(* Logix 5000 project; controller new_PLC_1 vendor 1 type 14 code 235 rev 37.11; software revision 37.00 *)

TASK MainTask (continuous, watchdog 500 ms) : MainProgram
TASK SafetyTask (periodic, rate 20 ms, priority 10, watchdog 20 ms, safety) : SafetyProgram

MODULES
   Local : vendor 1 type 14 code 235 (5069 0, rev 37.11)
      Tarjeta_Ethernet : vendor 1 type 12 code 200 (Ethernet 10.12.143.10, rev 10.7, Output RPI 10 ms)
         PLC_Safety : vendor 1 type 14 code 148 (ICP 1, rev 31.11, $66e82ebd$ RPI 20 ms)
         @7686e93b@:Partner : vendor 1 type 14 code 146 (ICP 2, rev 31.11)
      Variador_Conveyor_1 : PowerFlex 525-EENET (Ethernet 10.12.143.6, rev 5.1, Output RPI 20 ms)
      Camera_Conveyor_1 : vendor 678 type 100 code 260 (Ethernet 10.12.143.5, rev 12.1, Output RPI 60 ms)
      Point_IO_Gabinete_1 : 1734-AENTR (Ethernet 10.12.143.40, rev 5.12, Output RPI 20 ms)
         Modulo_Input_11 : 1734-IB8 (PointIO 1, rev 3.22)
              Point_IO_Gabinete_1:1:I.0   // Sensor Axis X -
              Point_IO_Gabinete_1:1:I.1   // Sensor Axis X +
              Point_IO_Gabinete_1:1:I.2   // Sensor Gripper Turn Conveyor
              Point_IO_Gabinete_1:1:I.3   // Sensor Gripper Close
              Point_IO_Gabinete_1:1:I.4   // Sensor Gripper Turn Storage
              Point_IO_Gabinete_1:1:I.5   // Sensor Axis Y -
              Point_IO_Gabinete_1:1:I.6   // Sensor Axis Y +
              Point_IO_Gabinete_1:1:I.7   // Sensor Gripper Open
              Point_IO_Gabinete_1:1:I   // Storage 1 Inputs
         Modulo_Input_12 : 1734-IB8 (PointIO 2, rev 3.22)
         Modulo_Output_11 : 1734-OB8 (PointIO 3, rev 3.22)
              Point_IO_Gabinete_1:3:O.0   // Axis X +
              Point_IO_Gabinete_1:3:O.1   // Axis X -
              Point_IO_Gabinete_1:3:O.2   // Gripper Close
              Point_IO_Gabinete_1:3:O.3   // Gripper Open
              Point_IO_Gabinete_1:3:O.4   // Gripper Turn Conveyor
              Point_IO_Gabinete_1:3:O.5   // Gripper Turn Storage
              Point_IO_Gabinete_1:3:O.6   // Axis Y +
              Point_IO_Gabinete_1:3:O.7   // Axis Y -
              Point_IO_Gabinete_1:3:O   // Storage 1 Outputs
         Modulo_Output_12 : 1734-OB8 (PointIO 4, rev 3.22)
              Point_IO_Gabinete_1:4:O.0   // Stack Light Blue
              Point_IO_Gabinete_1:4:O.1   // Stack Light Green
              Point_IO_Gabinete_1:4:O.2   // Stack Light Orange
              Point_IO_Gabinete_1:4:O.3   // Stack Light Red
              Point_IO_Gabinete_1:4:O   // Storage 1 Outputs Stack Lights
         Modulo_Relay_1 : 1734-OW4 (PointIO 5, rev 3.22)
      Point_IO_Gabinete_3 : 1734-AENTR (Ethernet 10.12.143.42, rev 5.12, Output RPI 20 ms)
         Modulo_Input_31 : 1734-IB8 (PointIO 1, rev 3.22)
         Modulo_Input_32 : 1734-IB8 (PointIO 2, rev 3.22)
         Modulo_Input_33 : 1734-IB8 (PointIO 3, rev 3.22)
              Point_IO_Gabinete_3:3:I.4   // Sensor Lane Change 2 +
              Point_IO_Gabinete_3:3:I.6   // Sensor Lane Change 1 +
              Point_IO_Gabinete_3:3:I.2   // Piston 1 retraido conveyor 1
              Point_IO_Gabinete_3:3:I.3   // Piston 1 activado conveyor 1
              Point_IO_Gabinete_3:3:I   // Sensors Lane Change +
         Modulo_Input_34 : 1734-IB8 (PointIO 4, rev 3.22)
              Point_IO_Gabinete_3:4:I.0   // Sensor Lane Change 1 -
              Point_IO_Gabinete_3:4:I.4   // Sensor Lane Change 2 -
              Point_IO_Gabinete_3:4:I   // Sensors Lane Change -
         Modulo_Input_35 : 1734-IB8 (PointIO 5, rev 3.22)
              Point_IO_Gabinete_3:5:I.0   // Inductive Sensor 1
              Point_IO_Gabinete_3:5:I.1   // Inductive Sensor 6
              Point_IO_Gabinete_3:5:I.2   // Inductive Sensor 5
              Point_IO_Gabinete_3:5:I.3   // Inductive Sensor 4
              Point_IO_Gabinete_3:5:I.4   // Inductive Sensor 3
              Point_IO_Gabinete_3:5:I.5   // Inductive Sensor 2
              Point_IO_Gabinete_3:5:I   // Conveyor 1 Inductive Sensors
         Modulo_Input_36 : 1734-IB8 (PointIO 6, rev 3.22)
         Modulo_Output_31 : 1734-OB8 (PointIO 7, rev 3.22)
              Point_IO_Gabinete_3:7:O.0   // Pneumatic Cylinder 0
              Point_IO_Gabinete_3:7:O.1   // Pneumatic Cylinder 1
              Point_IO_Gabinete_3:7:O.2   // Pneumatic Cylinder 2
              Point_IO_Gabinete_3:7:O.3   // Pneumatic Cylinder 3
              Point_IO_Gabinete_3:7:O.4   // Pneumatic Cylinder 4
              Point_IO_Gabinete_3:7:O.5   // Pneumatic Cylinder D
              Point_IO_Gabinete_3:7:O.6   // Lane Change 2
              Point_IO_Gabinete_3:7:O.7   // Lane Change 1
              Point_IO_Gabinete_3:7:O   // Conveyor 1 Pneumatic Cylinders
         Modulo_Output_32 : 1734-OB8 (PointIO 8, rev 3.22)
              Point_IO_Gabinete_3:8:O.0   // Main Valve
              Point_IO_Gabinete_3:8:O.2   // Cognex Light 2
              Point_IO_Gabinete_3:8:O.3   // Cognex Light 1
              Point_IO_Gabinete_3:8:O   // Main Valve
         Modulo_Relay_31 : 1734-OW4 (PointIO 9, rev 3.22)
         Modulo_Relay_32 : 1734-OW4 (PointIO 10, rev 3.22)
      PLC2 : vendor 1 type 14 code 235 (Ethernet 10.12.143.18, rev 37.11, $66dc2b48$ RPI 20 ms)
END_MODULES

VAR_GLOBAL   (* controller tags *)
   Data_from_PLC_2 : DINT[20];
   Data_From_PLC_Safety : DINT[20] := ([1] := 128);
        [0].11   // Pieza 1 puesta
        [0].12   // Pieza 2 puesta
        [0].13   // Pieza 3 puesta
        [0].14   // Pieza1 dejada
        [0].15   // Pieza 2 dejada
        [0].17   // Pieza 3 dejada
   Data_to_PLC_2 : DINT[20]; {produced}
        [0].0   // PB_START CONVEYORS DE PLC1 Y PLC2
        [1].0   // Pieza 1 etapa 1 salida y recorrido
        [1].1   // Pieza 1 etapa 2 foto cognex
        [1].2   // Pieza 1 etapa 3 listo para recolección
        [1].5   // Pieza 2 etapa 2 foto cognex
        [1].6   // Pieza 2 etapa 3 listo para recolección
        [1].8   // Pieza 3 etapa 2 foto cognex
        [1].7   // Pieza 3 etapa 1 salida y recorrido
        [1].4   // Pieza 2 etapa 1 salida y recorrido
        [1].9   // Pieza 3 etapa 3 listo para recolección
   Data_To_PLC_Safety : DINT[20] := ([0] := 16777216); {produced}
        [19].0   // Dato para mandar el trigger
   Fanuc_Strobe : BOOL;
   Height_1 : BOOL;
   Height_2 : BOOL;
   Height_3 : BOOL;
   Height_4 : BOOL;
   Height_5 : BOOL;
   Height_6 : BOOL;
   Height_Conveyor_1 : BOOL;
   Height_Conveyor_2 : BOOL;
   Process_1_Reset : ALIAS FOR Point_IO_Gabinete_1:2:I.6;   // Push Button Process 1 Reset
   Safety_OK : BOOL;
   Sensor_Height_1 : BOOL;
   Sensor_Height_2 : BOOL;
   Sensor_Height_3 : BOOL;
   Sensor_Height_4 : BOOL;
   Sensor_Height_5 : BOOL;
   Sensor_Height_6 : BOOL;
   Sensor_Height_Conveyor_1 : BOOL;
   Sensor_Height_Conveyor_2 : BOOL;
   Storage_On : BOOL;
END_VAR

PROGRAM MainProgram   (* main routine MainRoutine *)
VAR
   cleaning : BOOL;
   Counter_1 : COUNTER := (PRE := 3);
   Height_4_Number_2 : BOOL;
   Height_5_Number_2 : BOOL;
   Height_6_Number_2 : BOOL;
   HMI_Conveyor_OFF : BOOL;
   HMI_Conveyor_ON : BOOL;
   HMI_Fcognex1 : BOOL := 1;
   HMI_Fpowerflex1 : BOOL;
   HMI_Gripper_Close : BOOL;
   HMI_Gripper_Open : BOOL;
   HMI_Height_4_1 : BOOL;
   HMI_Height_4_2 : BOOL;
   HMI_Height_5_1 : BOOL;
   HMI_Height_5_2 : BOOL;
   HMI_Height_6_1 : BOOL;
   HMI_Height_6_2 : BOOL;
   HMI_Lane_Change_1 : BOOL;
   HMI_Lane_Change_2 : BOOL;
   HMI_Pneumatic_Cylinder_0 : BOOL;
   HMI_Pneumatic_Cylinder_1 : BOOL;
   HMI_Pneumatic_Cylinder_2 : BOOL;
   HMI_Pneumatic_Cylinder_3 : BOOL;
   HMI_Pneumatic_Cylinder_4 : BOOL;
   HMi_Screen_Storage1 : BOOL := 1;
   HMI_Turn_Conveyor : BOOL;
   HMI_Turn_Storage : BOOL;
   HMI_Y_Negative : BOOL;
   HMI_Y_Positive : BOOL;
   Pieza : COUNTER := (PRE := 3);
   Pieza_Detectada : BOOL;
   Pneumatic_Cylinder_0 : ALIAS FOR Point_IO_Gabinete_3:7:O.0;
   Recieve_bit_From_FANUC : BOOL;
   Reset_manual : BOOL;
   Send_Bit_to_FANUC_1 : BOOL;
   Send_Bit_to_FANUC_2 : BOOL;
   Send_Bit_to_FANUC_3 : BOOL;
   Send_Bit_to_FANUC_4 : BOOL;
   Sensor_Height_4_Number_2 : BOOL;
   Sensor_Height_5_Number_2 : BOOL;
   Sensor_Height_6_Number_2 : BOOL;
   Start_Button_1 : BOOL;
   Start_Button_2 : BOOL;
   Start_Button_3 : BOOL;
   Start_Conveyor1 : BOOL;
   Start_Robot_Fanuc : BOOL;
   Step_000 : SFC_STEP := (Status := 16#0020_0000, PauseTimer := 1);
   Step_001 : SFC_STEP := (Status := 16#0020_0000, PauseTimer := 1);
   Tiempo_ciclo : TIMER := (PRE := 1000000);
   Timer1 : TIMER := (PRE := 1000);
   Timer2 : TIMER := (PRE := 1000);
   Timer3 : TIMER := (PRE := 15000);
   Timer4 : TIMER := (PRE := 2000);
   Timer5 : TIMER := (PRE := 2000);
   Timer6 : TIMER := (PRE := 1000);
   Timer7 : TIMER := (PRE := 2000);
   Timer8 : TIMER := (PRE := 2000);
   timer_counter_1 : TIMER := (PRE := 2000);
   Timer_trigger : TIMER := (PRE := 3000);
   Tran_000 : BOOL;
   Tran_001 : BOOL;
   Trigger_Cognex_3 : BOOL;
END_VAR

ROUTINE E_Stop   (* ladder *)
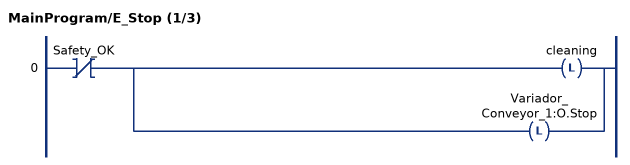
   0: XIO(Safety_OK)[OTL(cleaning) ,OTL(Variador_Conveyor_1:O.Stop) ];
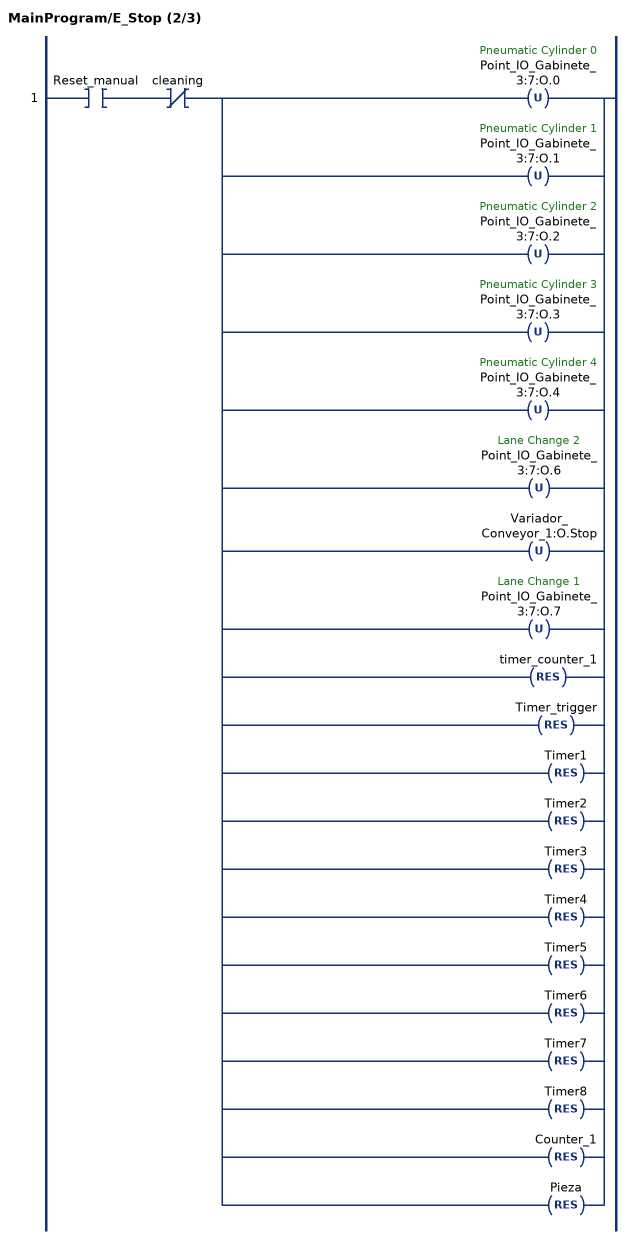
   1: XIC(Reset_manual)XIO(cleaning)[OTU(Point_IO_Gabinete_3:7:O.0) ,OTU(Point_IO_Gabinete_3:7:O.1) ,OTU(Point_IO_Gabinete_3:7:O.2) ,OTU(Point_IO_Gabinete_3:7:O.3) ,OTU(Point_IO_Gabinete_3:7:O.4) ,OTU(Point_IO_Gabinete_3:7:O.6) ,OTU(Variador_Conveyor_1:O.Stop) ,OTU(Point_IO_Gabinete_3:7:O.7) ,RES(timer_counter_1) ,RES(Timer_trigger) ,RES(Timer1) ,RES(Timer2) ,RES(Timer3) ,RES(Timer4) ,RES(Timer5) ,RES(Timer6) ,RES(Timer7) ,RES(Timer8) ,RES(Counter_1) ,RES(Pieza) ];
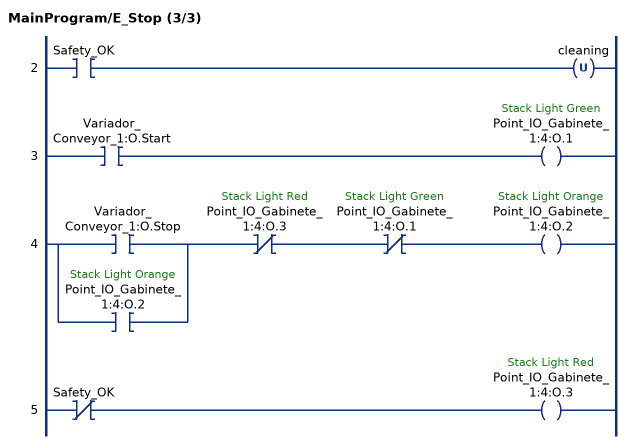
   2: XIC(Safety_OK)OTU(cleaning);
   3: XIC(Variador_Conveyor_1:O.Start)OTE(Point_IO_Gabinete_1:4:O.1);
   4: [XIC(Variador_Conveyor_1:O.Stop) ,XIC(Point_IO_Gabinete_1:4:O.2) ]XIO(Point_IO_Gabinete_1:4:O.3)XIO(Point_IO_Gabinete_1:4:O.1)OTE(Point_IO_Gabinete_1:4:O.2);
   5: XIO(Safety_OK)OTE(Point_IO_Gabinete_1:4:O.3);
END_ROUTINE

ROUTINE MainRoutine   (* ladder *)
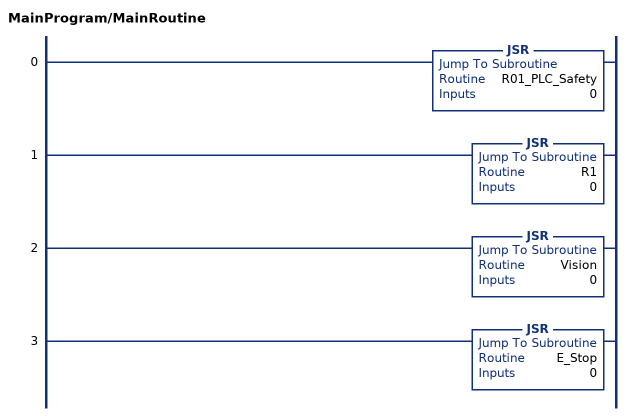
   0: JSR(R01_PLC_Safety,0);
   1: JSR(R1,0);
   2: JSR(Vision,0);
   3: JSR(E_Stop,0);
END_ROUTINE

ROUTINE R01_PLC_Safety   (* ladder *)
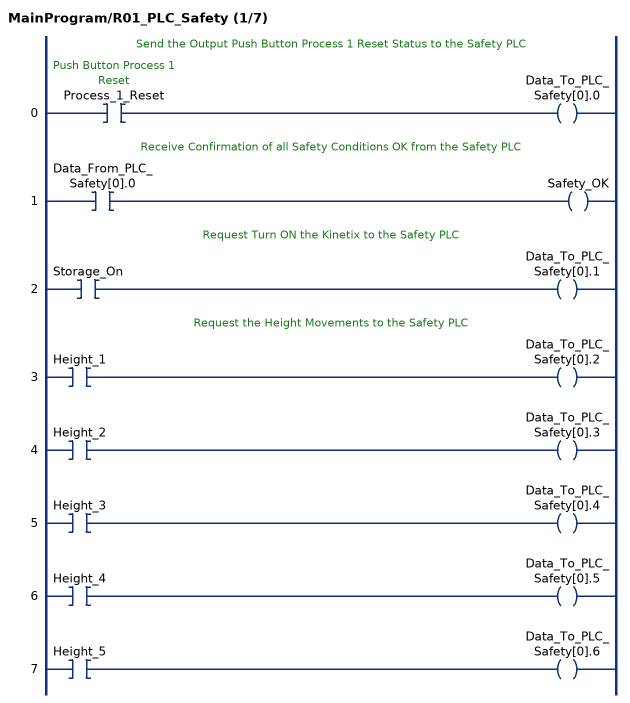
   // Send the Output Push Button Process 1 Reset Status to the Safety PLC
   0: XIC(Process_1_Reset)OTE(Data_To_PLC_Safety[0].0);
   // Receive Confirmation of all Safety Conditions OK from the Safety PLC
   1: XIC(Data_From_PLC_Safety[0].0)OTE(Safety_OK);
   // Request Turn ON the Kinetix to the Safety PLC
   2: XIC(Storage_On)OTE(Data_To_PLC_Safety[0].1);
   // Request the Height Movements to the Safety PLC
   3: XIC(Height_1)OTE(Data_To_PLC_Safety[0].2);
   4: XIC(Height_2)OTE(Data_To_PLC_Safety[0].3);
   5: XIC(Height_3)OTE(Data_To_PLC_Safety[0].4);
   6: XIC(Height_4)OTE(Data_To_PLC_Safety[0].5);
   7: XIC(Height_5)OTE(Data_To_PLC_Safety[0].6);
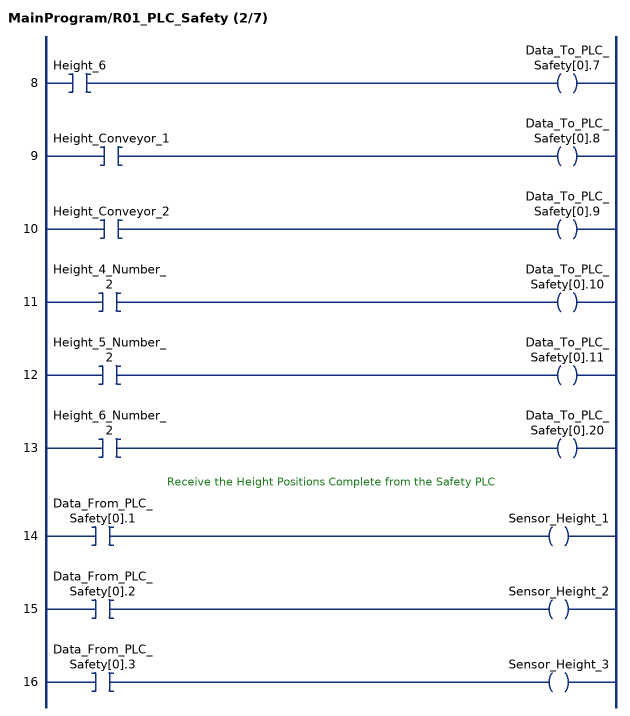
   8: XIC(Height_6)OTE(Data_To_PLC_Safety[0].7);
   9: XIC(Height_Conveyor_1)OTE(Data_To_PLC_Safety[0].8);
   10: XIC(Height_Conveyor_2)OTE(Data_To_PLC_Safety[0].9);
   11: XIC(Height_4_Number_2)OTE(Data_To_PLC_Safety[0].10);
   12: XIC(Height_5_Number_2)OTE(Data_To_PLC_Safety[0].11);
   13: XIC(Height_6_Number_2)OTE(Data_To_PLC_Safety[0].20);
   // Receive the Height Positions Complete from the Safety PLC
   14: XIC(Data_From_PLC_Safety[0].1)OTE(Sensor_Height_1);
   15: XIC(Data_From_PLC_Safety[0].2)OTE(Sensor_Height_2);
   16: XIC(Data_From_PLC_Safety[0].3)OTE(Sensor_Height_3);
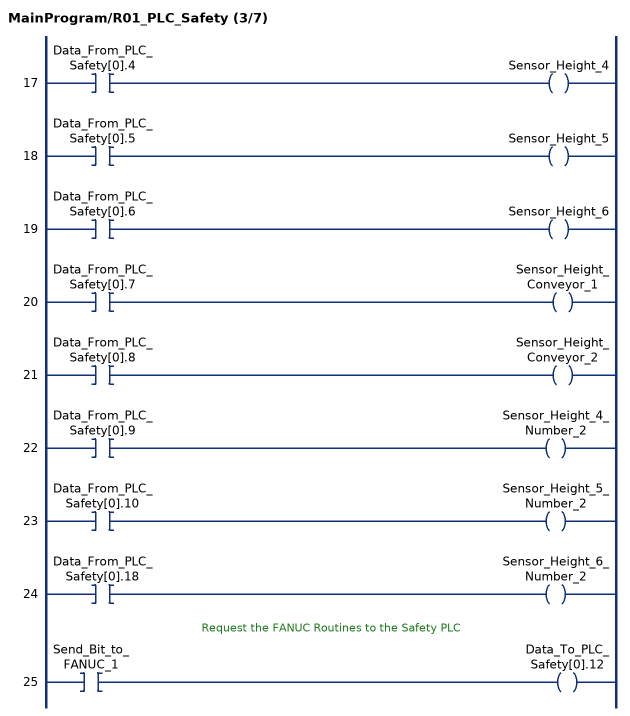
   17: XIC(Data_From_PLC_Safety[0].4)OTE(Sensor_Height_4);
   18: XIC(Data_From_PLC_Safety[0].5)OTE(Sensor_Height_5);
   19: XIC(Data_From_PLC_Safety[0].6)OTE(Sensor_Height_6);
   20: XIC(Data_From_PLC_Safety[0].7)OTE(Sensor_Height_Conveyor_1);
   21: XIC(Data_From_PLC_Safety[0].8)OTE(Sensor_Height_Conveyor_2);
   22: XIC(Data_From_PLC_Safety[0].9)OTE(Sensor_Height_4_Number_2);
   23: XIC(Data_From_PLC_Safety[0].10)OTE(Sensor_Height_5_Number_2);
   24: XIC(Data_From_PLC_Safety[0].18)OTE(Sensor_Height_6_Number_2);
   // Request the FANUC Routines to the Safety PLC
   25: XIC(Send_Bit_to_FANUC_1)OTE(Data_To_PLC_Safety[0].12);
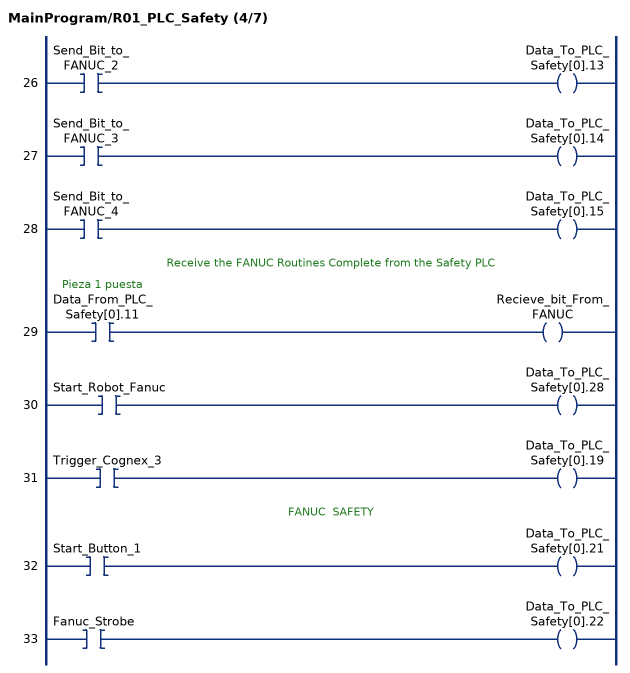
   26: XIC(Send_Bit_to_FANUC_2)OTE(Data_To_PLC_Safety[0].13);
   27: XIC(Send_Bit_to_FANUC_3)OTE(Data_To_PLC_Safety[0].14);
   28: XIC(Send_Bit_to_FANUC_4)OTE(Data_To_PLC_Safety[0].15);
   // Receive the FANUC Routines Complete from the Safety PLC
   29: XIC(Data_From_PLC_Safety[0].11)OTE(Recieve_bit_From_FANUC);
   30: XIC(Start_Robot_Fanuc)OTE(Data_To_PLC_Safety[0].28);
   31: XIC(Trigger_Cognex_3)OTE(Data_To_PLC_Safety[0].19);
   // FANUC  SAFETY
   32: XIC(Start_Button_1)OTE(Data_To_PLC_Safety[0].21);
   33: XIC(Fanuc_Strobe)OTE(Data_To_PLC_Safety[0].22);
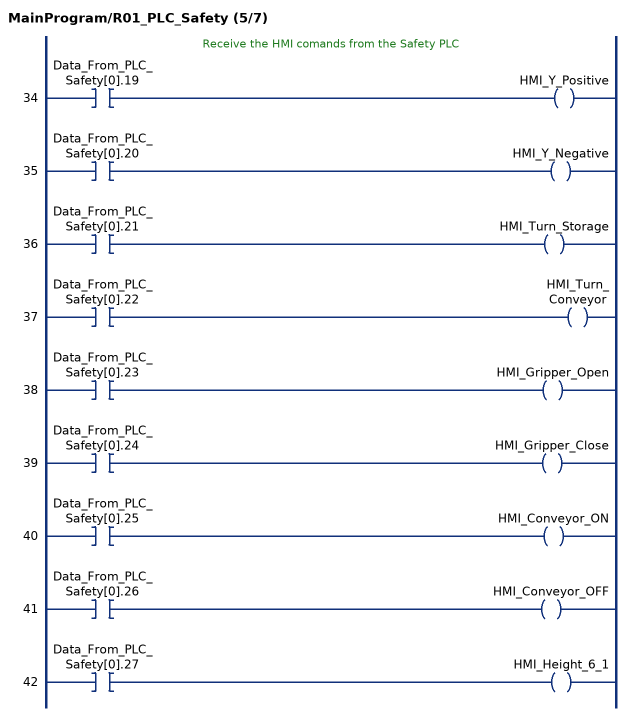
   // Receive the HMI comands from the Safety PLC
   34: XIC(Data_From_PLC_Safety[0].19)OTE(HMI_Y_Positive);
   35: XIC(Data_From_PLC_Safety[0].20)OTE(HMI_Y_Negative);
   36: XIC(Data_From_PLC_Safety[0].21)OTE(HMI_Turn_Storage);
   37: XIC(Data_From_PLC_Safety[0].22)OTE(HMI_Turn_Conveyor);
   38: XIC(Data_From_PLC_Safety[0].23)OTE(HMI_Gripper_Open);
   39: XIC(Data_From_PLC_Safety[0].24)OTE(HMI_Gripper_Close);
   40: XIC(Data_From_PLC_Safety[0].25)OTE(HMI_Conveyor_ON);
   41: XIC(Data_From_PLC_Safety[0].26)OTE(HMI_Conveyor_OFF);
   42: XIC(Data_From_PLC_Safety[0].27)OTE(HMI_Height_6_1);
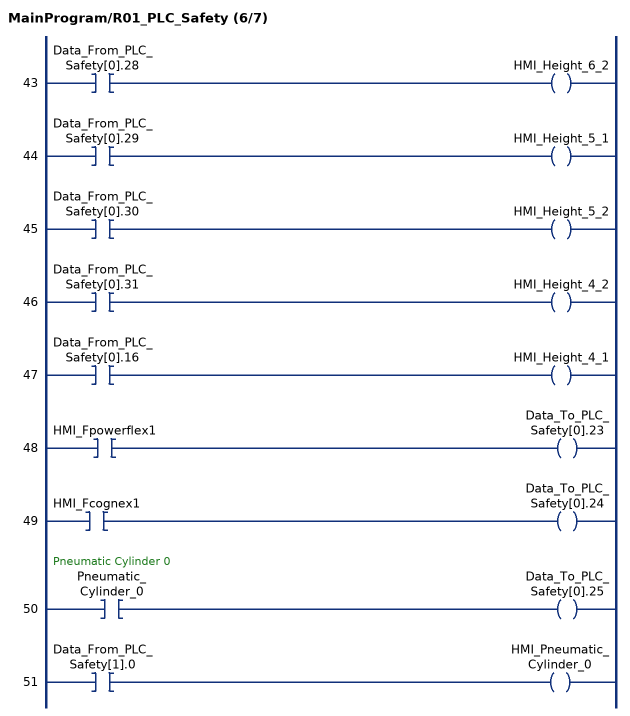
   43: XIC(Data_From_PLC_Safety[0].28)OTE(HMI_Height_6_2);
   44: XIC(Data_From_PLC_Safety[0].29)OTE(HMI_Height_5_1);
   45: XIC(Data_From_PLC_Safety[0].30)OTE(HMI_Height_5_2);
   46: XIC(Data_From_PLC_Safety[0].31)OTE(HMI_Height_4_2);
   47: XIC(Data_From_PLC_Safety[0].16)OTE(HMI_Height_4_1);
   48: XIC(HMI_Fpowerflex1)OTE(Data_To_PLC_Safety[0].23);
   49: XIC(HMI_Fcognex1)OTE(Data_To_PLC_Safety[0].24);
   50: XIC(Pneumatic_Cylinder_0)OTE(Data_To_PLC_Safety[0].25);
   51: XIC(Data_From_PLC_Safety[1].0)OTE(HMI_Pneumatic_Cylinder_0);
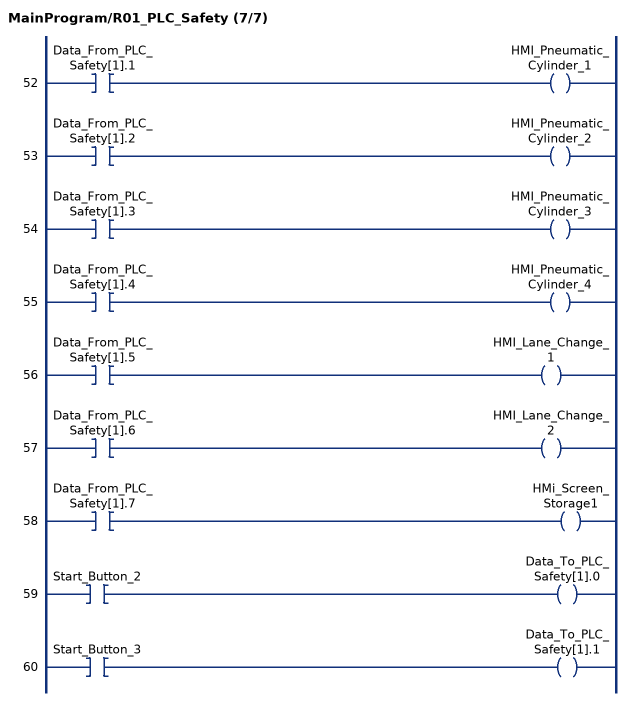
   52: XIC(Data_From_PLC_Safety[1].1)OTE(HMI_Pneumatic_Cylinder_1);
   53: XIC(Data_From_PLC_Safety[1].2)OTE(HMI_Pneumatic_Cylinder_2);
   54: XIC(Data_From_PLC_Safety[1].3)OTE(HMI_Pneumatic_Cylinder_3);
   55: XIC(Data_From_PLC_Safety[1].4)OTE(HMI_Pneumatic_Cylinder_4);
   56: XIC(Data_From_PLC_Safety[1].5)OTE(HMI_Lane_Change_1);
   57: XIC(Data_From_PLC_Safety[1].6)OTE(HMI_Lane_Change_2);
   58: XIC(Data_From_PLC_Safety[1].7)OTE(HMi_Screen_Storage1);
   59: XIC(Start_Button_2)OTE(Data_To_PLC_Safety[1].0);
   60: XIC(Start_Button_3)OTE(Data_To_PLC_Safety[1].1);
END_ROUTINE

ROUTINE R1   (* ladder *)
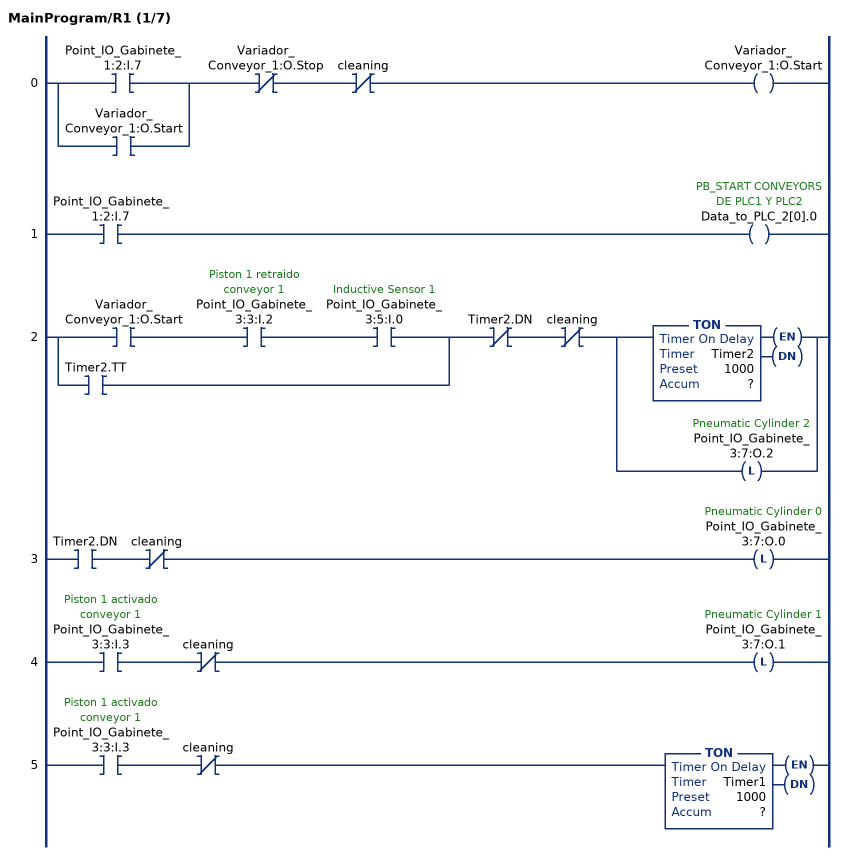
   0: [XIC(Point_IO_Gabinete_1:2:I.7) ,XIC(Variador_Conveyor_1:O.Start) ]XIO(Variador_Conveyor_1:O.Stop)XIO(cleaning)OTE(Variador_Conveyor_1:O.Start);
   1: XIC(Point_IO_Gabinete_1:2:I.7)OTE(Data_to_PLC_2[0].0);
   2: [XIC(Variador_Conveyor_1:O.Start) XIC(Point_IO_Gabinete_3:3:I.2) XIC(Point_IO_Gabinete_3:5:I.0) ,XIC(Timer2.TT) ]XIO(Timer2.DN)XIO(cleaning)[TON(Timer2,?,?) ,OTL(Point_IO_Gabinete_3:7:O.2) ];
   3: XIC(Timer2.DN)XIO(cleaning)OTL(Point_IO_Gabinete_3:7:O.0);
   4: XIC(Point_IO_Gabinete_3:3:I.3)XIO(cleaning)OTL(Point_IO_Gabinete_3:7:O.1);
   5: XIC(Point_IO_Gabinete_3:3:I.3)XIO(cleaning)TON(Timer1,?,?);
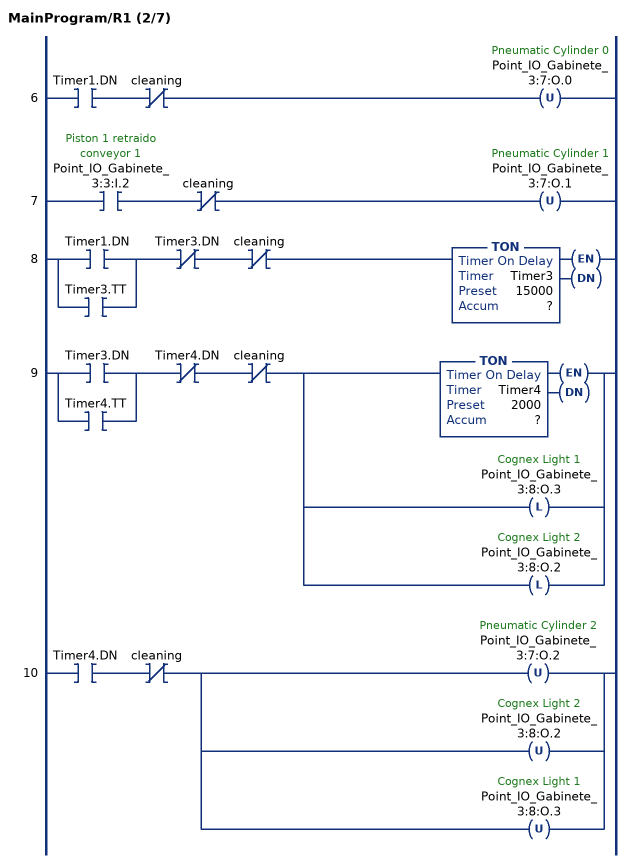
   6: XIC(Timer1.DN)XIO(cleaning)OTU(Point_IO_Gabinete_3:7:O.0);
   7: XIC(Point_IO_Gabinete_3:3:I.2)XIO(cleaning)OTU(Point_IO_Gabinete_3:7:O.1);
   8: [XIC(Timer1.DN) ,XIC(Timer3.TT) ]XIO(Timer3.DN)XIO(cleaning)TON(Timer3,?,?);
   9: [XIC(Timer3.DN) ,XIC(Timer4.TT) ]XIO(Timer4.DN)XIO(cleaning)[TON(Timer4,?,?) ,OTL(Point_IO_Gabinete_3:8:O.3) ,OTL(Point_IO_Gabinete_3:8:O.2) ];
   10: XIC(Timer4.DN)XIO(cleaning)[OTU(Point_IO_Gabinete_3:7:O.2) ,OTU(Point_IO_Gabinete_3:8:O.2) ,OTU(Point_IO_Gabinete_3:8:O.3) ];
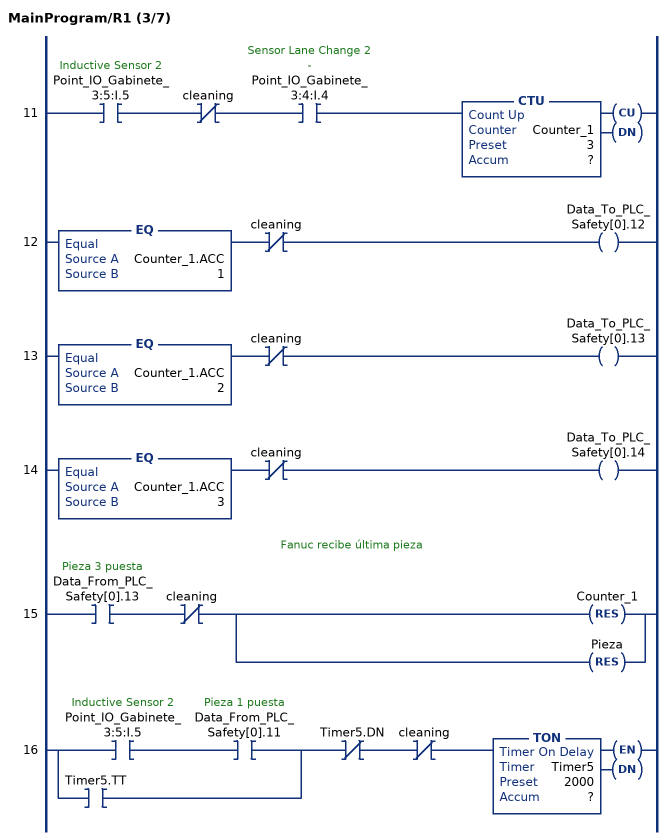
   11: XIC(Point_IO_Gabinete_3:5:I.5)XIO(cleaning)XIC(Point_IO_Gabinete_3:4:I.4)CTU(Counter_1,?,?);
   12: EQ(Counter_1.ACC,1)XIO(cleaning)OTE(Data_To_PLC_Safety[0].12);
   13: EQ(Counter_1.ACC,2)XIO(cleaning)OTE(Data_To_PLC_Safety[0].13);
   14: EQ(Counter_1.ACC,3)XIO(cleaning)OTE(Data_To_PLC_Safety[0].14);
   // Fanuc recibe última pieza
   15: XIC(Data_From_PLC_Safety[0].13)XIO(cleaning)[RES(Counter_1) ,RES(Pieza) ];
   16: [XIC(Point_IO_Gabinete_3:5:I.5) XIC(Data_From_PLC_Safety[0].11) ,XIC(Timer5.TT) ]XIO(Timer5.DN)XIO(cleaning)TON(Timer5,?,?);
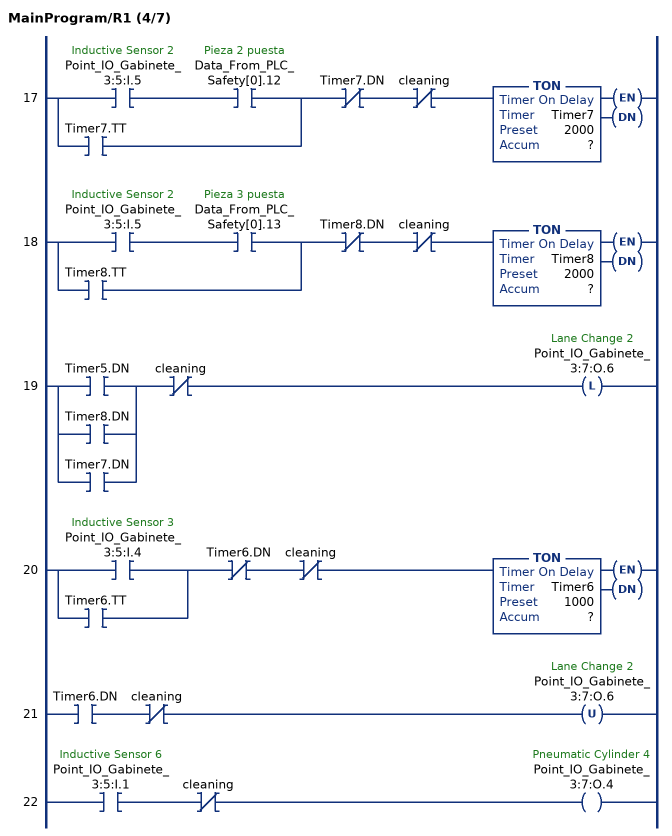
   17: [XIC(Point_IO_Gabinete_3:5:I.5) XIC(Data_From_PLC_Safety[0].12) ,XIC(Timer7.TT) ]XIO(Timer7.DN)XIO(cleaning)TON(Timer7,?,?);
   18: [XIC(Point_IO_Gabinete_3:5:I.5) XIC(Data_From_PLC_Safety[0].13) ,XIC(Timer8.TT) ]XIO(Timer8.DN)XIO(cleaning)TON(Timer8,?,?);
   19: [XIC(Timer5.DN) ,XIC(Timer8.DN) ,XIC(Timer7.DN) ]XIO(cleaning)OTL(Point_IO_Gabinete_3:7:O.6);
   20: [XIC(Point_IO_Gabinete_3:5:I.4) ,XIC(Timer6.TT) ]XIO(Timer6.DN)XIO(cleaning)TON(Timer6,?,?);
   21: XIC(Timer6.DN)XIO(cleaning)OTU(Point_IO_Gabinete_3:7:O.6);
   22: XIC(Point_IO_Gabinete_3:5:I.1)XIO(cleaning)OTE(Point_IO_Gabinete_3:7:O.4);
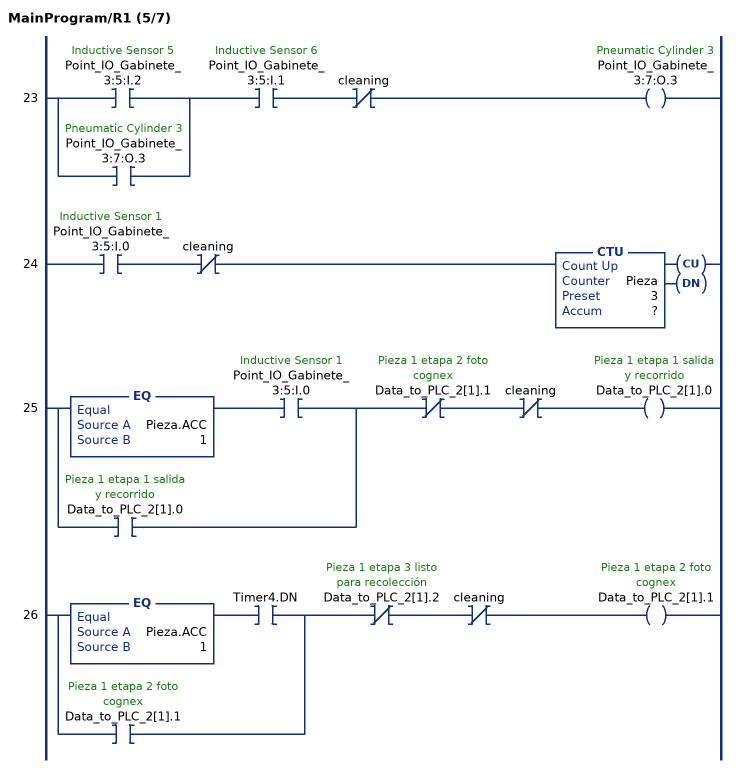
   23: [XIC(Point_IO_Gabinete_3:5:I.2) ,XIC(Point_IO_Gabinete_3:7:O.3) ]XIC(Point_IO_Gabinete_3:5:I.1)XIO(cleaning)OTE(Point_IO_Gabinete_3:7:O.3);
   24: XIC(Point_IO_Gabinete_3:5:I.0)XIO(cleaning)CTU(Pieza,?,?);
   25: [EQ(Pieza.ACC,1) XIC(Point_IO_Gabinete_3:5:I.0) ,XIC(Data_to_PLC_2[1].0) ]XIO(Data_to_PLC_2[1].1)XIO(cleaning)OTE(Data_to_PLC_2[1].0);
   26: [EQ(Pieza.ACC,1) XIC(Timer4.DN) ,XIC(Data_to_PLC_2[1].1) ]XIO(Data_to_PLC_2[1].2)XIO(cleaning)OTE(Data_to_PLC_2[1].1);
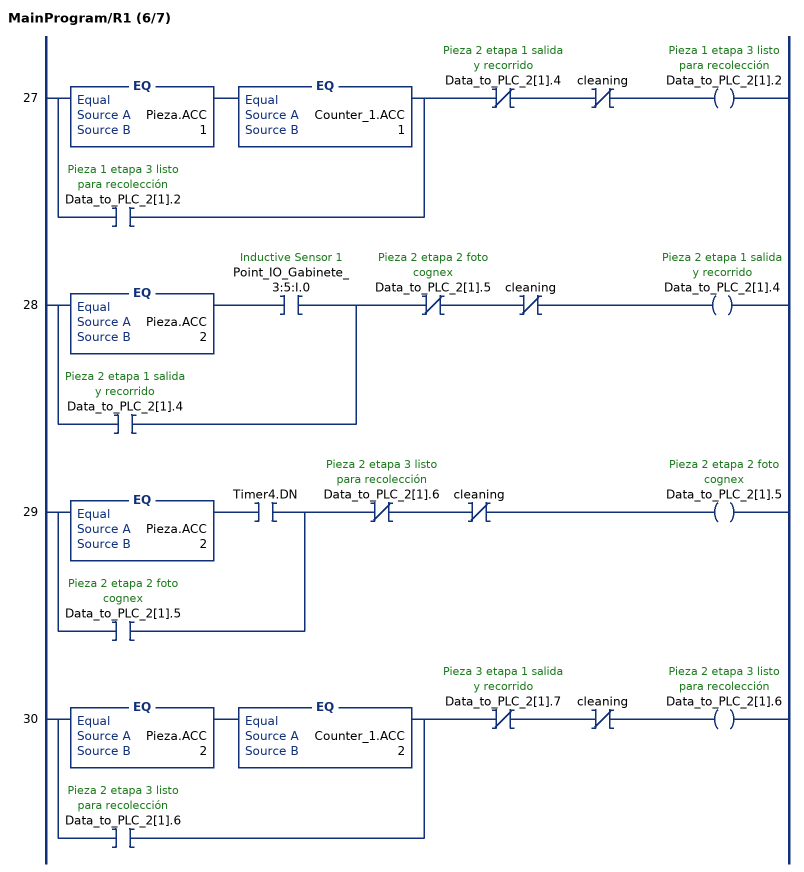
   27: [EQ(Pieza.ACC,1) EQ(Counter_1.ACC,1) ,XIC(Data_to_PLC_2[1].2) ]XIO(Data_to_PLC_2[1].4)XIO(cleaning)OTE(Data_to_PLC_2[1].2);
   28: [EQ(Pieza.ACC,2) XIC(Point_IO_Gabinete_3:5:I.0) ,XIC(Data_to_PLC_2[1].4) ]XIO(Data_to_PLC_2[1].5)XIO(cleaning)OTE(Data_to_PLC_2[1].4);
   29: [EQ(Pieza.ACC,2) XIC(Timer4.DN) ,XIC(Data_to_PLC_2[1].5) ]XIO(Data_to_PLC_2[1].6)XIO(cleaning)OTE(Data_to_PLC_2[1].5);
   30: [EQ(Pieza.ACC,2) EQ(Counter_1.ACC,2) ,XIC(Data_to_PLC_2[1].6) ]XIO(Data_to_PLC_2[1].7)XIO(cleaning)OTE(Data_to_PLC_2[1].6);
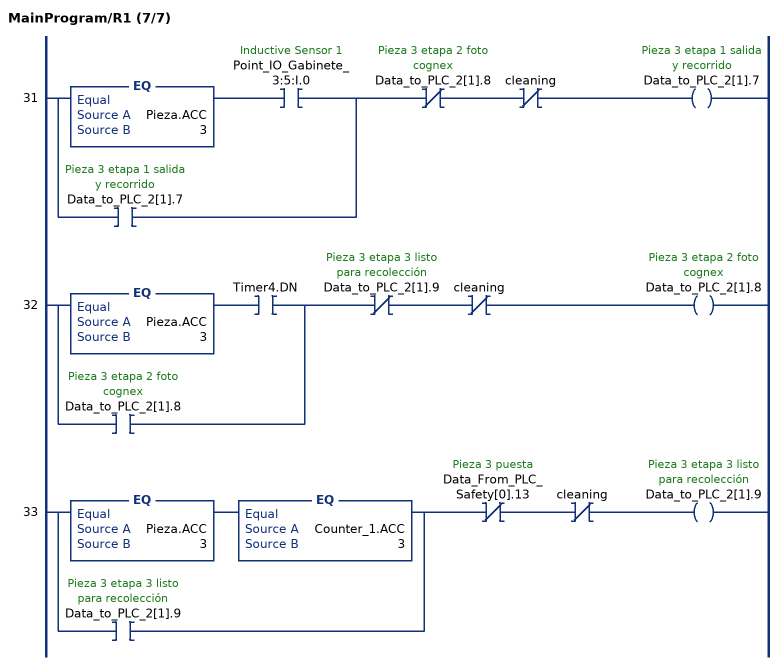
   31: [EQ(Pieza.ACC,3) XIC(Point_IO_Gabinete_3:5:I.0) ,XIC(Data_to_PLC_2[1].7) ]XIO(Data_to_PLC_2[1].8)XIO(cleaning)OTE(Data_to_PLC_2[1].7);
   32: [EQ(Pieza.ACC,3) XIC(Timer4.DN) ,XIC(Data_to_PLC_2[1].8) ]XIO(Data_to_PLC_2[1].9)XIO(cleaning)OTE(Data_to_PLC_2[1].8);
   33: [EQ(Pieza.ACC,3) EQ(Counter_1.ACC,3) ,XIC(Data_to_PLC_2[1].9) ]XIO(Data_From_PLC_Safety[0].13)XIO(cleaning)OTE(Data_to_PLC_2[1].9);
END_ROUTINE

ROUTINE Vision   (* ladder *)
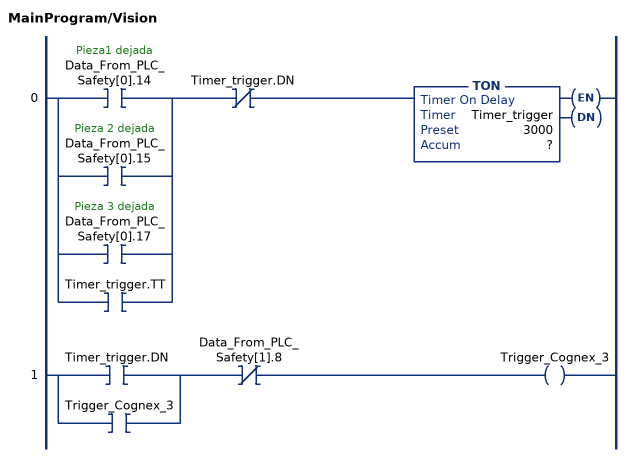
   0: [XIC(Data_From_PLC_Safety[0].14) ,XIC(Data_From_PLC_Safety[0].15) ,XIC(Data_From_PLC_Safety[0].17) ,XIC(Timer_trigger.TT) ]XIO(Timer_trigger.DN)TON(Timer_trigger,?,?);
   1: [XIC(Timer_trigger.DN) ,XIC(Trigger_Cognex_3) ]XIO(Data_From_PLC_Safety[1].8)OTE(Trigger_Cognex_3);
END_ROUTINE
END_PROGRAM

PROGRAM SafetyProgram   (* main routine MainRoutine, safety *)

ROUTINE MainRoutine   (* ladder *)
END_ROUTINE
END_PROGRAM
